// TIA Portal V21 export
DATA_BLOCK "Pompapistoni_Timer"   // DB25
{ S7_Optimized_Access := 'TRUE' }
// stored: MemoryReserve 100
   VAR
      RitardoPartenza { S7_SetPoint := 'True'} : "Std_stTimer";   // AttesaRampa
      RitardoInAllarme { S7_SetPoint := 'True'} : "Std_stTimer";   // Tempo in cui si può discostare
   END_VAR
BEGIN
   RitardoPartenza.IN := FALSE;
   RitardoPartenza.O := FALSE;
   RitardoPartenza.Preset := 10.0;
   RitardoPartenza.TempoTrascorso := 0.0;
   RitardoInAllarme.IN := FALSE;
   RitardoInAllarme.O := FALSE;
   RitardoInAllarme.Preset := 3.0;
   RitardoInAllarme.TempoTrascorso := 0.0;
END_DATA_BLOCK
